METHOD  getNewCandy :REFERENCE TO AbstractCandy
VAR_INPUT
	(*preferred candy type, it must be a pure candy type *)
	candyType	:CandyTypes;
END_VAR
VAR
	(* the __NEW operator requires a stricktly typed pointer *)
	alpenliebe			:POINTER TO Alpenliebe;		
	(* the __NEW operator requires a stricktly typed pointer *)
	altoids				:POINTER TO Altoids;
	(* the __NEW operator requires a stricktly typed pointer *)
	bobsStripes			:POINTER TO BobsSweetStripes;
	(* the __NEW operator requires a stricktly typed pointer *)
	candyCorn			:POINTER TO BrachsCandyCorn;
	(* the __NEW operator requires a stricktly typed pointer *)
	chupChups			:POINTER TO ChupaChups;
	(* the __NEW operator requires a stricktly typed pointer *)
	goldbears			:POINTER TO Goldbears;
	(* the __NEW operator requires a stricktly typed pointer *)
	mAndMs				:POINTER TO MnMs;	
	(* the __NEW operator requires a stricktly typed pointer *)
	skittles			:POINTER TO SkittlesSour;
	(* the __NEW operator requires a stricktly typed pointer *)
	poppins				:POINTER TO Poppins;
	(* the __NEW operator requires a stricktly typed pointer *)
	snickers			:POINTER TO SnickersBar;
	(* the __NEW operator requires a stricktly typed pointer *)
	twizzlers			:POINTER TO TwizzlersLicorizeTwists;
	(* the __NEW operator requires a stricktly typed pointer *)
	gobstopper			:POINTER TO WonkaGobstopper;
	(* return value is just a candy *)
	candy				:POINTER TO AbstractCandy;
END_VAR
getNewCandy REF= 0;
RETURN(THIS^.isCandyTypeInvalidForMachine(candyType));

CASE candyType OF
CandyTypes.CANDY_BARS:
	snickers := __NEW(SnickersBar());
	candy := snickers;
CandyTypes.CANDY_CORN:
	candyCorn := __NEW(BrachsCandyCorn());
	candy := candyCorn;
CandyTypes.CANDY_STICKS:
	bobsStripes := __NEW(BobsSweetStripes());
	candy := bobsStripes;
CandyTypes.CARAMEL_CANDY:
	alpenliebe := __NEW(Alpenliebe());
	candy := alpenliebe;
CandyTypes.CHOCOLATE_CANDY:
	mAndMs := __NEW(MnMs());
	candy := mAndMs;
CandyTypes.GUMMY_CANDY:;		
	goldbears := __NEW(Goldbears());
	candy := goldbears;		
CandyTypes.HARD_CANDY:
	poppins := __NEW(Poppins());
	candy := poppins;		
CandyTypes.LOLLIPOPS:
	chupChups := __NEW(ChupaChups());
	candy := chupChups;
CandyTypes.JAWBREAKERS:
	gobstopper := __NEW(WonkaGobstopper());
	candy := gobstopper;
CandyTypes.LICORICE_CANDY:
	twizzlers := __NEW(TwizzlersLicorizeTwists());
	candy := twizzlers;
CandyTypes.MINTS:
	altoids := __NEW(Altoids());
	candy := altoids;
CandyTypes.SOUR_CANDY:
	skittles := __NEW(SkittlesSour());
	candy := skittles;
ELSE
	RETURN;	
END_CASE

RETURN(candy <= 0);
getNewCandy REF= candy^;
END_METHOD

END_FUNCTION_BLOCK

// ---- Candies/Classes/Goldbears.TcPOU
(*

short summary
=============
A specialized candy. It can be consumed by any candy consumer.
It supports dynamic creation. Furthermore, it calls the method 
AbstractCandy.initializeDispatchers after FB_init.

legal notes
===========
SPDX-FileCopyrightText: © 2024 ekvip automation GmbH <info@ekvip.de>
SPDX-License-Identifier: Apache-2.0
For details check: Apache-2.0_

.. _Apache-2.0: https://www.apache.org/licenses/LICENSE-2.0

*)

{attribute 'enable_dynamic_creation'}
{attribute 'call_after_init'}
FUNCTION_BLOCK FINAL Goldbears EXTENDS AbstractCandy
VAR_INPUT
END_VAR
VAR_OUTPUT
END_VAR
VAR
END_VAR

(*

short summary
=============
it initializes the amount, the candy name and 
the binary coded candy type  

legal notes
===========
SPDX-FileCopyrightText: © 2024 ekvip automation GmbH <info@ekvip.de>
SPDX-License-Identifier: Apache-2.0
For details check: Apache-2.0_

.. _Apache-2.0: https://www.apache.org/licenses/LICENSE-2.0

*)

METHOD FB_init :BOOL
VAR_INPUT
	(* if TRUE, the retain variables are initialized (warm start / cold start) *)
	bInitRetains	:BOOL;
	(* if TRUE, the instance afterwards gets moved into the copy code (online change) *)
	bInCopyCode		:BOOL;
END_VAR
THIS^.amount := 75;
THIS^.name := 'HARIBO Goldbears';
THIS^.candyType := CandyTypes.GUMMY_CANDY;
END_METHOD

END_FUNCTION_BLOCK

// ---- Candies/Classes/MnMs.TcPOU
(*

short summary
=============
A specialized candy. It can be consumed by any candy consumer.
It supports dynamic creation. Furthermore, it calls the method 
AbstractCandy.initializeDispatchers after FB_init.

legal notes
===========
SPDX-FileCopyrightText: © 2024 ekvip automation GmbH <info@ekvip.de>
SPDX-License-Identifier: Apache-2.0
For details check: Apache-2.0_

.. _Apache-2.0: https://www.apache.org/licenses/LICENSE-2.0

*)

{attribute 'enable_dynamic_creation'}
{attribute 'call_after_init'}
FUNCTION_BLOCK FINAL MnMs EXTENDS AbstractCandy
VAR_INPUT
END_VAR
VAR_OUTPUT
END_VAR
VAR
END_VAR

(*

short summary
=============
it initializes the amount, the candy name and 
the binary coded candy type  

legal notes
===========
SPDX-FileCopyrightText: © 2024 ekvip automation GmbH <info@ekvip.de>
SPDX-License-Identifier: Apache-2.0
For details check: Apache-2.0_

.. _Apache-2.0: https://www.apache.org/licenses/LICENSE-2.0

*)

METHOD FB_init :BOOL
VAR_INPUT
	(* if TRUE, the retain variables are initialized (warm start / cold start) *)
	bInitRetains	:BOOL;
	(* if TRUE, the instance afterwards gets moved into the copy code (online change) *)
	bInCopyCode		:BOOL;
END_VAR
THIS^.amount := 45;
THIS^.name := 'M&M$'s';
THIS^.candyType := CandyTypes.CHOCOLATE_CANDY;
END_METHOD

END_FUNCTION_BLOCK

// ---- Candies/Classes/Poppins.TcPOU
(*

short summary
=============
A specialized candy. It can be consumed by any candy consumer.
It supports dynamic creation. Furthermore, it calls the method 
AbstractCandy.initializeDispatchers after FB_init.

legal notes
===========
SPDX-FileCopyrightText: © 2024 ekvip automation GmbH <info@ekvip.de>
SPDX-License-Identifier: Apache-2.0
For details check: Apache-2.0_

.. _Apache-2.0: https://www.apache.org/licenses/LICENSE-2.0

*)

{attribute 'enable_dynamic_creation'}
{attribute 'call_after_init'}
FUNCTION_BLOCK FINAL Poppins EXTENDS AbstractCandy
VAR_INPUT
END_VAR
VAR_OUTPUT
END_VAR
VAR
END_VAR

(*

short summary
=============
it initializes the amount, the candy name and 
the binary coded candy type  

legal notes
===========
SPDX-FileCopyrightText: © 2024 ekvip automation GmbH <info@ekvip.de>
SPDX-License-Identifier: Apache-2.0
For details check: Apache-2.0_

.. _Apache-2.0: https://www.apache.org/licenses/LICENSE-2.0

*)

METHOD FB_init :BOOL
VAR_INPUT
	(* if TRUE, the retain variables are initialized (warm start / cold start) *)
	bInitRetains	:BOOL;
	(* if TRUE, the instance afterwards gets moved into the copy code (online change) *)
	bInCopyCode		:BOOL;
END_VAR
THIS^.amount := 18;
THIS^.name := 'Parle Poppins';
THIS^.candyType := CandyTypes.HARD_CANDY;
END_METHOD

END_FUNCTION_BLOCK

// ---- NinjaMonkeys/Classes/IndividualCandyPreferences.TcPOU
(*

short summary
=============
This abstraction is to define different preferences for all types of candies 

legal notes
===========
SPDX-FileCopyrightText: © 2024 ekvip automation GmbH <info@ekvip.de>
SPDX-License-Identifier: Apache-2.0
For details check: Apache-2.0_

.. _Apache-2.0: https://www.apache.org/licenses/LICENSE-2.0

*)

FUNCTION_BLOCK ABSTRACT IndividualCandyPreferences
VAR
END_VAR

(*

short summary
=============
This method is to get the tastiness for a given candy type

legal notes
===========
SPDX-FileCopyrightText: © 2024 ekvip automation GmbH <info@ekvip.de>
SPDX-License-Identifier: Apache-2.0
For details check: Apache-2.0_

.. _Apache-2.0: https://www.apache.org/licenses/LICENSE-2.0

*)
METHOD ABSTRACT howIsTheCandy :TasteScale
VAR_INPUT
	(* candy type to get the tastiness for it *)
	candyType :CandyTypes;
END_VAR
END_METHOD

END_FUNCTION_BLOCK

// ---- NinjaCandyBehavior/Classes/PickyNinjaCandyBehavior.TcPOU
(*

short summary
=============
the behavior of a picky ninja

legal notes
===========
SPDX-FileCopyrightText: © 2024 ekvip automation GmbH <info@ekvip.de>
SPDX-License-Identifier: Apache-2.0
For details check: Apache-2.0_

.. _Apache-2.0: https://www.apache.org/licenses/LICENSE-2.0

*)

FUNCTION_BLOCK PickyNinjaCandyBehavior EXTENDS AbstractNinjaCandyConsumeBehavior
VAR_STAT
	(* default provider for the pickies*)
	pickyDefaultProvider :NinjaIncCandyMachineProvider(ConsumerTypes.PICKY);
END_VAR

(*

short summary
=============
This method calculates the satisfaction level
for a candy eating picky consumer.

legal notes
===========
SPDX-FileCopyrightText: © 2024 ekvip automation GmbH <info@ekvip.de>
SPDX-License-Identifier: Apache-2.0
For details check: Apache-2.0_

.. _Apache-2.0: https://www.apache.org/licenses/LICENSE-2.0

*)

METHOD  calculateSatisfactionLevel
VAR_INPUT
	(* taste scale of candy *)
	tastiness				:TasteScale;
	(* amount of the candies to eat *)
	amountOfCandy			:CandyAmountInGram;
END_VAR
VAR_IN_OUT
	(* the satisfaction level of the consumer *)
	actualSatisfactionLevel	:SatisfactionLevelInPercent;
END_VAR
VAR
	(* the greedy consumer likes everything *)
	pickyScale :DINT;
END_VAR
VAR CONSTANT
	(* maximum possible satisfaction level*)
	MAX_SATISFACTION 		:SatisfactionLevelInPercent := 100;
	(* it is a lower limit as it is named *)
	AVOID_DIVISON_BY_ZERO 	:SatisfactionLevelInPercent := 1;
	(* factor for the greediness of the consumer *)
	GREEDINESS				:SatisfactionLevelInPercent := 80;
	(* for one a candy package the maximum amount *)
	MAX_AMOUNT				:CandyAmountInGram := 500;
END_VAR
RETURN(actualSatisfactionLevel >= MAX_SATISFACTION);
RETURN(tastiness = TasteScale.OKAY);
pickyScale := tastiness;

{warning disable C0196}
{warning disable C0197}
actualSatisfactionLevel := TO_UINT(
	actualSatisfactionLevel + TO_SINT(
		LN(
			TO_REAL(MAX_SATISFACTION)
			/LIMIT(AVOID_DIVISON_BY_ZERO, actualSatisfactionLevel, MAX_SATISFACTION)
		) * (
			TO_REAL(amountOfCandy)
			/TO_REAL(MAX_AMOUNT)
		)
		* (MAX_SATISFACTION - GREEDINESS)
		* pickyScale
	)
);
{warning restore C0196}
{warning restore C0197}
END_METHOD

(*

short summary
=============
inject the candy vending machine provider
during declaration.

legal notes
===========
SPDX-FileCopyrightText: © 2024 ekvip automation GmbH <info@ekvip.de>
SPDX-License-Identifier: Apache-2.0
For details check: Apache-2.0_

.. _Apache-2.0: https://www.apache.org/licenses/LICENSE-2.0

*)

METHOD FB_init :BOOL
VAR_INPUT
	(* if TRUE, the retain variables are initialized (warm start / cold start) *)
	bInitRetains		:BOOL;
	(* if TRUE, the instance afterwards gets moved into the copy code (online change) *)
	bInCopyCode			:BOOL;
	(* candy vending machine provider for the consumer *)
	candyMachineProvider:REFERENCE TO CandyMachineProvider;
END_VAR
IF (__ISVALIDREF(candyMachineProvider)) THEN
	THIS^.candyMachineProvider REF= candyMachineProvider;
ELSE
	THIS^.candyMachineProvider REF= THIS^.pickyDefaultProvider;
END_IF
END_METHOD

END_FUNCTION_BLOCK

// ---- NinjaMonkeys/Classes/AjninsCandyPreferences.TcPOU
(*

short summary
=============
Ajnins candy preferences

legal notes
===========
SPDX-FileCopyrightText: © 2024 ekvip automation GmbH <info@ekvip.de>
SPDX-License-Identifier: Apache-2.0
For details check: Apache-2.0_

.. _Apache-2.0: https://www.apache.org/licenses/LICENSE-2.0

*)

FUNCTION_BLOCK FINAL AjninsCandyPreferences EXTENDS IndividualCandyPreferences
VAR
END_VAR

(*

short summary
=============
This method is to get the tastiness for a given candy type

legal notes
===========
SPDX-FileCopyrightText: © 2024 ekvip automation GmbH <info@ekvip.de>
SPDX-License-Identifier: Apache-2.0
For details check: Apache-2.0_

.. _Apache-2.0: https://www.apache.org/licenses/LICENSE-2.0

*)
METHOD howIsTheCandy :TasteScale
VAR_INPUT
	(* candy type to get the tastiness for it *)
	candyType	:CandyTypes;
END_VAR
CASE candyType OF
CandyTypes.CANDY_BARS:
	howIsTheCandy := TasteScale.DELICIOUS;
CandyTypes.CANDY_CORN:
	howIsTheCandy := TasteScale.DISGUSTING;
CandyTypes.CANDY_STICKS:
	howIsTheCandy := TasteScale.DELICIOUS;
CandyTypes.CARAMEL_CANDY:
	howIsTheCandy := TasteScale.OKAY;
CandyTypes.CHOCOLATE_CANDY:
	howIsTheCandy := TasteScale.OKAY;
CandyTypes.GUMMY_CANDY:
	howIsTheCandy := TasteScale.DISGUSTING;
CandyTypes.HARD_CANDY:
	howIsTheCandy := TasteScale.DISGUSTING;
CandyTypes.JAWBREAKERS:
	howIsTheCandy := TasteScale.DELICIOUS;
CandyTypes.LICORICE_CANDY:
	howIsTheCandy := TasteScale.DISGUSTING;
CandyTypes.LOLLIPOPS:
	howIsTheCandy := TasteScale.DELICIOUS;
CandyTypes.MINTS:
	howIsTheCandy := TasteScale.DISGUSTING;
CandyTypes.SOUR_CANDY:;
	howIsTheCandy := TasteScale.DELICIOUS;
ELSE
	howIsTheCandy := TasteScale.OKAY;
END_CASE
END_METHOD

END_FUNCTION_BLOCK

// ---- NinjaMonkeys/Classes/NinjaMonkey.TcPOU
(*

short summary
=============
A ninja candy consumer. It can eat candies and the
candies will effect the satisfaction of the consumer.
Since ninjas a heterogeneous crowd is it necessary to inject
the ninjas behavior.

legal notes
===========
SPDX-FileCopyrightText: © 2024 ekvip automation GmbH <info@ekvip.de>
SPDX-License-Identifier: Apache-2.0
For details check: Apache-2.0_

.. _Apache-2.0: https://www.apache.org/licenses/LICENSE-2.0

*)

{attribute 'reflection'}
FUNCTION_BLOCK FINAL NinjaMonkey EXTENDS AbstractCandyConsumer
VAR
	(* the candy consume behavior of the ninja instance *) 
	candyBehavior				:REFERENCE TO AbstractNinjaCandyConsumeBehavior;
	(* candy preferences of the ninja *)
	candyPreferences			:REFERENCE TO IndividualCandyPreferences;
	(* ninjas name is the instance path without the project nodes *)
	{attribute 'instance-path'}
	{attribute 'no-init'}
	myName						:ConsumerName;
END_VAR
VAR_STAT
	(* default behavior for ninja monkeys *)
	defaultCandyBehavior		:CommonNinjaCandyBehavior(0);
END_VAR

(*

short summary
=============
method to eat candy bars

legal notes
===========
SPDX-FileCopyrightText: © 2024 ekvip automation GmbH <info@ekvip.de>
SPDX-License-Identifier: Apache-2.0
For details check: Apache-2.0_

.. _Apache-2.0: https://www.apache.org/licenses/LICENSE-2.0

*)

METHOD  eatCandyBars
VAR_INPUT
	(* amount of candy that the consumer eats in gram *)
	amount	:CandyAmountInGram;
END_VAR
THIS^.candyBehavior.calculateSatisfactionLevel(THIS^.getTastiness(CandyTypes.CANDY_BARS), amount, THIS^.satisfaction);
END_METHOD

(*

short summary
=============
method to eat candy corn

legal notes
===========
SPDX-FileCopyrightText: © 2024 ekvip automation GmbH <info@ekvip.de>
SPDX-License-Identifier: Apache-2.0
For details check: Apache-2.0_

.. _Apache-2.0: https://www.apache.org/licenses/LICENSE-2.0

*)

METHOD  eatCandyCorn
VAR_INPUT
	(* amount of candy that the consumer eats in gram *)
	amount	:CandyAmountInGram;
END_VAR
THIS^.candyBehavior.calculateSatisfactionLevel(THIS^.getTastiness(CandyTypes.CANDY_CORN), amount, THIS^.satisfaction);
END_METHOD

(*

short summary
=============
method to eat candy sticks

legal notes
===========
SPDX-FileCopyrightText: © 2024 ekvip automation GmbH <info@ekvip.de>
SPDX-License-Identifier: Apache-2.0
For details check: Apache-2.0_

.. _Apache-2.0: https://www.apache.org/licenses/LICENSE-2.0

*)

METHOD  eatCandySticks
VAR_INPUT
	(* amount of candy that the consumer eats in gram *)
	amount	:CandyAmountInGram;
END_VAR
THIS^.candyBehavior.calculateSatisfactionLevel(THIS^.getTastiness(CandyTypes.CANDY_STICKS), amount, THIS^.satisfaction);
END_METHOD

(*

short summary
=============
method to eat caramel candy

legal notes
===========
SPDX-FileCopyrightText: © 2024 ekvip automation GmbH <info@ekvip.de>
SPDX-License-Identifier: Apache-2.0
For details check: Apache-2.0_

.. _Apache-2.0: https://www.apache.org/licenses/LICENSE-2.0

*)

METHOD  eatCaramelCandy
VAR_INPUT
	(* amount of candy that the consumer eats in gram *)
	amount	:CandyAmountInGram;
END_VAR
THIS^.candyBehavior.calculateSatisfactionLevel(THIS^.getTastiness(CandyTypes.CARAMEL_CANDY), amount, THIS^.satisfaction);
END_METHOD

(*

short summary
=============
method to eat choclate candy

legal notes
===========
SPDX-FileCopyrightText: © 2024 ekvip automation GmbH <info@ekvip.de>
SPDX-License-Identifier: Apache-2.0
For details check: Apache-2.0_

.. _Apache-2.0: https://www.apache.org/licenses/LICENSE-2.0

*)

METHOD  eatChoclateCandy
VAR_INPUT
	(* amount of candy that the consumer eats in gram *)
	amount	:CandyAmountInGram;
END_VAR
THIS^.candyBehavior.calculateSatisfactionLevel(THIS^.getTastiness(CandyTypes.CHOCOLATE_CANDY), amount, THIS^.satisfaction);
END_METHOD

(*

short summary
=============
method to eat gummy candy

legal notes
===========
SPDX-FileCopyrightText: © 2024 ekvip automation GmbH <info@ekvip.de>
SPDX-License-Identifier: Apache-2.0
For details check: Apache-2.0_

.. _Apache-2.0: https://www.apache.org/licenses/LICENSE-2.0

*)

METHOD  eatGummyCandy
VAR_INPUT
	(* amount of candy that the consumer eats in gram *)
	amount	:CandyAmountInGram;
END_VAR
THIS^.candyBehavior.calculateSatisfactionLevel(THIS^.getTastiness(CandyTypes.GUMMY_CANDY), amount, THIS^.satisfaction);
END_METHOD

(*

short summary
=============
method to eat hard candy

legal notes
===========
SPDX-FileCopyrightText: © 2024 ekvip automation GmbH <info@ekvip.de>
SPDX-License-Identifier: Apache-2.0
For details check: Apache-2.0_

.. _Apache-2.0: https://www.apache.org/licenses/LICENSE-2.0

*)

METHOD  eatHardCandy
VAR_INPUT
	(* amount of candy that the consumer eats in gram *)
	amount	:CandyAmountInGram;
END_VAR
THIS^.candyBehavior.calculateSatisfactionLevel(THIS^.getTastiness(CandyTypes.HARD_CANDY), amount, THIS^.satisfaction);
END_METHOD

(*

short summary
=============
method to eat jawbrakers

legal notes
===========
SPDX-FileCopyrightText: © 2024 ekvip automation GmbH <info@ekvip.de>
SPDX-License-Identifier: Apache-2.0
For details check: Apache-2.0_

.. _Apache-2.0: https://www.apache.org/licenses/LICENSE-2.0

*)

METHOD  eatJawbreakers
VAR_INPUT
	(* amount of candy that the consumer eats in gram *)
	amount	:CandyAmountInGram;
END_VAR
THIS^.candyBehavior.calculateSatisfactionLevel(THIS^.getTastiness(CandyTypes.JAWBREAKERS), amount, THIS^.satisfaction);
END_METHOD

(*

short summary
=============
method to eat licorice candy

legal notes
===========
SPDX-FileCopyrightText: © 2024 ekvip automation GmbH <info@ekvip.de>
SPDX-License-Identifier: Apache-2.0
For details check: Apache-2.0_

.. _Apache-2.0: https://www.apache.org/licenses/LICENSE-2.0

*)

METHOD  eatLicoriceCandy
VAR_INPUT
	(* amount of candy that the consumer eats in gram *)
	amount	:CandyAmountInGram;
END_VAR
THIS^.candyBehavior.calculateSatisfactionLevel(THIS^.getTastiness(CandyTypes.LICORICE_CANDY), amount, THIS^.satisfaction);
END_METHOD

(*

short summary
=============
method to eat lollipops

legal notes
===========
SPDX-FileCopyrightText: © 2024 ekvip automation GmbH <info@ekvip.de>
SPDX-License-Identifier: Apache-2.0
For details check: Apache-2.0_

.. _Apache-2.0: https://www.apache.org/licenses/LICENSE-2.0

*)

METHOD  eatLollipops
VAR_INPUT
	(* amount of candy that the consumer eats in gram *)
	amount	:CandyAmountInGram;
END_VAR
THIS^.candyBehavior.calculateSatisfactionLevel(THIS^.getTastiness(CandyTypes.LOLLIPOPS), amount, THIS^.satisfaction);
END_METHOD

(*

short summary
=============
method to eat mints

legal notes
===========
SPDX-FileCopyrightText: © 2024 ekvip automation GmbH <info@ekvip.de>
SPDX-License-Identifier: Apache-2.0
For details check: Apache-2.0_

.. _Apache-2.0: https://www.apache.org/licenses/LICENSE-2.0

*)

METHOD  eatMints
VAR_INPUT
	(* amount of candy that the consumer eats in gram *)
	amount	:CandyAmountInGram;
END_VAR
THIS^.candyBehavior.calculateSatisfactionLevel(THIS^.getTastiness(CandyTypes.MINTS), amount, THIS^.satisfaction);
END_METHOD

(*

short summary
=============
method to eat sour candy

legal notes
===========
SPDX-FileCopyrightText: © 2024 ekvip automation GmbH <info@ekvip.de>
SPDX-License-Identifier: Apache-2.0
For details check: Apache-2.0_

.. _Apache-2.0: https://www.apache.org/licenses/LICENSE-2.0

*)

METHOD  eatSourCandy
VAR_INPUT
	(* amount of candy that the consumer eats in gram *)
	amount	:CandyAmountInGram;
END_VAR
THIS^.candyBehavior.calculateSatisfactionLevel(THIS^.getTastiness(CandyTypes.SOUR_CANDY), amount, THIS^.satisfaction);
END_METHOD

(*

short summary
=============
it sets the candy consume behavior and remove the project nodes from name

legal notes
===========
SPDX-FileCopyrightText: © 2024 ekvip automation GmbH <info@ekvip.de>
SPDX-License-Identifier: Apache-2.0
For details check: Apache-2.0_

.. _Apache-2.0: https://www.apache.org/licenses/LICENSE-2.0

*)

METHOD FB_init : BOOL
VAR_INPUT
	(* if TRUE, the retain variables are initialized (warm start / cold start) *)
	bInitRetains		:BOOL;
	(* if TRUE, the instance afterwards gets moved into the copy code (online change) *)
	bInCopyCode			:BOOL;
	(* the candy consume behavior of the ninja *)
	ninjaCandyBehavior	:REFERENCE TO AbstractNinjaCandyConsumeBehavior;
	(* candy preferences of the ninja *)
	candyPreferences	:REFERENCE TO IndividualCandyPreferences;
END_VAR
VAR CONSTANT
	(* numer of nodes to remove from name *)
	NUMBER_OF_PROJECT_NODES	:UINT := 2;
	(* for the path the node delimiter string *)
	INSTANCE_PATH_DELIMITER	:STRING(1) := '.';
END_VAR
IF (__ISVALIDREF(ninjaCandyBehavior)) THEN
	THIS^.candyBehavior REF= ninjaCandyBehavior;
ELSE
	THIS^.candyBehavior REF= THIS^.defaultCandyBehavior;
END_IF
THIS^.candyPreferences REF= candyPreferences;
THIS^.removeNodesFromPath(THIS^.myName, NUMBER_OF_PROJECT_NODES, INSTANCE_PATH_DELIMITER);
END_METHOD

(*

short summary
=============
This method is just to deal with invalid
candy preferences, no preferences means everthing is DELICIOUS

legal notes
===========
SPDX-FileCopyrightText: © 2024 ekvip automation GmbH <info@ekvip.de>
SPDX-License-Identifier: Apache-2.0
For details check: Apache-2.0_

.. _Apache-2.0: https://www.apache.org/licenses/LICENSE-2.0

*)

METHOD PRIVATE getTastiness :TasteScale
VAR_INPUT
	candyType	:CandyTypes;
END_VAR
IF (__ISVALIDREF(THIS^.candyPreferences)) THEN
	getTastiness := THIS^.candyPreferences.howIsTheCandy(candyType);
ELSE
	getTastiness := TasteScale.DELICIOUS;
END_IF
END_METHOD

(*

short summary
=============
This is an api method to loot a candy vending machine with the consumer

legal notes
===========
SPDX-FileCopyrightText: © 2024 ekvip automation GmbH <info@ekvip.de>
SPDX-License-Identifier: Apache-2.0
For details check: Apache-2.0_

.. _Apache-2.0: https://www.apache.org/licenses/LICENSE-2.0

*)

METHOD lootCandies
VAR_INPUT
	(* rising edge strats the looting *)
	execute :BOOL;
END_VAR
VAR_INST
	(* to get the rising edge of the execute flag *)
	executionEdge	:Tc2_Standard.R_TRIG;
END_VAR
executionEdge(CLK := execute);
RETURN(NOT executionEdge.Q);
THIS^.candyBehavior.lootACandyMachine(THIS^, THIS^.candyPreferences);
END_METHOD

(*

short summary
=============
the instance path of the consumer without the project nodes

legal notes
===========
SPDX-FileCopyrightText: © 2024 ekvip automation GmbH <info@ekvip.de>
SPDX-License-Identifier: Apache-2.0
For details check: Apache-2.0_

.. _Apache-2.0: https://www.apache.org/licenses/LICENSE-2.0

*)

PROPERTY name :ConsumerName
GET
(*

short summary
=============
getter for the instance name of the object

legal notes
===========
SPDX-FileCopyrightText: © 2024 ekvip automation GmbH <info@ekvip.de>
SPDX-License-Identifier: Apache-2.0
For details check: Apache-2.0_

.. _Apache-2.0: https://www.apache.org/licenses/LICENSE-2.0

*)

VAR
END_VAR
name := THIS^.myName;
END_GET
END_PROPERTY

(*

short summary
=============
helper method to remove nodes from a path

legal notes
===========
SPDX-FileCopyrightText: © 2024 ekvip automation GmbH <info@ekvip.de>
SPDX-License-Identifier: Apache-2.0
For details check: Apache-2.0_

.. _Apache-2.0: https://www.apache.org/licenses/LICENSE-2.0

*)
{attribute 'estimated-stack-usage' := '4096'}
METHOD PRIVATE removeNodesFromPath
VAR_IN_OUT
	(* the path to remove the nodes from it *)
	path :Tc2_System.T_MaxString;
END_VAR
VAR_INPUT
	
	numberOfNodesToRemove	:UINT;
	delimiter				:STRING(1);
END_VAR
VAR
	found	:INT;
END_VAR
VAR CONSTANT
	NOTHING		:INT := 0;
	NO_NODES	:UINT:= 0;
END_VAR
RETURN (numberOfNodesToRemove <= NO_NODES);
found := Tc2_Standard.FIND(path, delimiter);
RETURN (found <= NOTHING);
path := RIGHT(path, LEN(path) - found);
THIS^.removeNodesFromPath(path, numberOfNodesToRemove-1, delimiter);
END_METHOD

END_FUNCTION_BLOCK

// ---- NinjaCandyBehavior/Classes/CommonNinjaCandyBehavior.TcPOU
(*

short summary
=============
the behavior of a common ninja

legal notes
===========
SPDX-FileCopyrightText: © 2024 ekvip automation GmbH <info@ekvip.de>
SPDX-License-Identifier: Apache-2.0
For details check: Apache-2.0_

.. _Apache-2.0: https://www.apache.org/licenses/LICENSE-2.0

*)

FUNCTION_BLOCK CommonNinjaCandyBehavior EXTENDS AbstractNinjaCandyConsumeBehavior

(*

short summary
=============
This method calculates the satisfaction level
for a candy eating usual consumer.

legal notes
===========
SPDX-FileCopyrightText: © 2024 ekvip automation GmbH <info@ekvip.de>
SPDX-License-Identifier: Apache-2.0
For details check: Apache-2.0_

.. _Apache-2.0: https://www.apache.org/licenses/LICENSE-2.0

*)

METHOD  calculateSatisfactionLevel
VAR_INPUT
	(* taste scale of candy *)
	tastiness				:TasteScale;
	(* amount of the candies to eat *)
	amountOfCandy			:CandyAmountInGram;
END_VAR
VAR_IN_OUT
	(* the satisfaction level of the consumer *)
	actualSatisfactionLevel	:SatisfactionLevelInPercent;
END_VAR
VAR
	(* the common consumer likes DELICIOUS and Okay *)
	pickyScale :DINT;
	(* relationship between actual and maximum satisfaction level *)
	statisfactionRelationship :REAL;
	gradient :REAL;
	(* relationship between given and maximum candy amaount *) 
	amountRelationship :REAL;
END_VAR
VAR CONSTANT
	(* maximum possible satisfaction level*)
	MAX_SATISFACTION 		:SatisfactionLevelInPercent := 100;
	(* it is a lower limit as it is named *)
	AVOID_DIVISON_BY_ZERO 	:SatisfactionLevelInPercent := 1;
	(* factor for the greediness of the consumer *)
	GREEDINESS				:SatisfactionLevelInPercent := 79;
	(* for one a candy package the maximum amount *)
	MAX_AMOUNT				:CandyAmountInGram := 500;
	(* between e and 10 *)
	LOGARITHM_BASE			:REAL := 6.359;
END_VAR
RETURN(actualSatisfactionLevel >= MAX_SATISFACTION);

pickyScale					:= SEL(tastiness = TasteScale.OKAY, tastiness, TasteScale.DELICIOUS);
statisfactionRelationship	:= TO_REAL(MAX_SATISFACTION)/LIMIT(AVOID_DIVISON_BY_ZERO, actualSatisfactionLevel, MAX_SATISFACTION);
gradient					:= LN(statisfactionRelationship)/LN(LOGARITHM_BASE);
amountRelationship			:= TO_REAL(amountOfCandy)/TO_REAL(MAX_AMOUNT);

{warning disable C0196}
{warning disable C0197}
actualSatisfactionLevel := TO_UINT(
	actualSatisfactionLevel + TO_SINT(
		gradient * amountRelationship * (MAX_SATISFACTION - GREEDINESS) * pickyScale
	)
);
{warning restore C0196}
{warning restore C0197}
END_METHOD

END_FUNCTION_BLOCK
